ABB RAPID module: Module1.mod

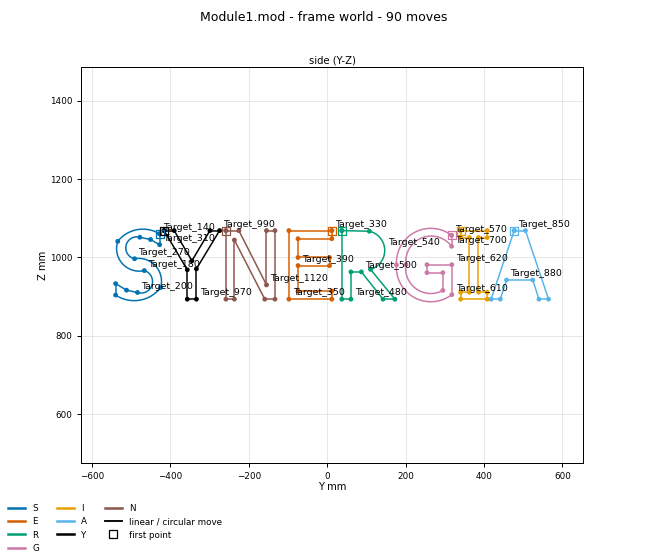
[picture p0: tool path of Module1.mod in frame world, 90 of 90 moves have a stored position in this frame; points joined in program order, loops and branches not executed]
MODULE Module1
	CONST robtarget Target_140:=[[750,-427.603905619,1060.300093764],[0,0,0.978993144,-0.20389317],[0,0,0,0],[9E9,9E9,9E9,9E9,9E9,9E9]];
	CONST robtarget Target_150:=[[750,-479.650096867,1071.645312565],[0,0,0.978993144,-0.20389317],[0,0,0,0],[9E9,9E9,9E9,9E9,9E9,9E9]];
	CONST robtarget Target_160:=[[750,-534.355323771,1041.137310133],[0,0,0.978993144,-0.20389317],[0,0,0,0],[9E9,9E9,9E9,9E9,9E9,9E9]];
	CONST robtarget Target_170:=[[750,-527.158200594,989.9597372],[0,0,0.978993144,-0.20389317],[0,0,0,0],[9E9,9E9,9E9,9E9,9E9,9E9]];
	CONST robtarget Target_180:=[[750,-466.603095246,966.560223424],[0,0,0.978993144,-0.20389317],[0,0,0,0],[9E9,9E9,9E9,9E9,9E9,9E9]];
	CONST robtarget Target_190:=[[750,-447.511219233,927.862391171],[0,0,0.978993144,-0.20389317],[0,0,0,0],[9E9,9E9,9E9,9E9,9E9,9E9]];
	CONST robtarget Target_200:=[[750,-484.046369152,910.543205595],[0,0,0.978993144,-0.20389317],[0,0,0,0],[9E9,9E9,9E9,9E9,9E9,9E9]];
	CONST robtarget Target_210:=[[750,-512.054878066,916.499445466],[0,0,0.978993144,-0.20389317],[0,0,0,0],[9E9,9E9,9E9,9E9,9E9,9E9]];
	CONST robtarget Target_220:=[[750,-539.77975651,933.233643197],[0,0,0.978993144,-0.20389317],[0,0,0,0],[9E9,9E9,9E9,9E9,9E9,9E9]];
	CONST robtarget Target_230:=[[750,-539.77975651,904.019704785],[0,0,0.978993144,-0.20389317],[0,0,0,0],[9E9,9E9,9E9,9E9,9E9,9E9]];
	CONST robtarget Target_240:=[[750,-482.344586332,890.405442224],[0,0,0.978993144,-0.20389317],[0,0,0,0],[9E9,9E9,9E9,9E9,9E9,9E9]];
	CONST robtarget Target_250:=[[750,-424.980323771,923.164761511],[0,0,0.978993144,-0.20389317],[0,0,0,0],[9E9,9E9,9E9,9E9,9E9,9E9]];
	CONST robtarget Target_260:=[[750,-439.941831064,980.617658594],[0,0,0.978993144,-0.20389317],[0,0,0,0],[9E9,9E9,9E9,9E9,9E9,9E9]];
	CONST robtarget Target_270:=[[750,-491.420761372,996.76686848],[0,0,0.978993144,-0.20389317],[0,0,0,0],[9E9,9E9,9E9,9E9,9E9,9E9]];
	CONST robtarget Target_280:=[[750,-511.753520692,1035.145616454],[0,0,0.978993144,-0.20389317],[0,0,0,0],[9E9,9E9,9E9,9E9,9E9,9E9]];
	CONST robtarget Target_290:=[[750,-478.090129282,1051.507549193],[0,0,0.978993144,-0.20389317],[0,0,0,0],[9E9,9E9,9E9,9E9,9E9,9E9]];
	CONST robtarget Target_300:=[[750,-450.719788925,1045.834939793],[0,0,0.978993144,-0.20389317],[0,0,0,0],[9E9,9E9,9E9,9E9,9E9,9E9]];
	CONST robtarget Target_310:=[[750,-427.603905619,1032.504307702],[0,0,0.978993144,-0.20389317],[0,0,0,0],[9E9,9E9,9E9,9E9,9E9,9E9]];
	CONST robtarget Target_320:=[[750,-427.603905619,1060.300093764],[0,0,0.978993144,-0.20389317],[0,0,0,0],[9E9,9E9,9E9,9E9,9E9,9E9]];
	CONST robtarget Target_330:=[[750,11.739692436,1068.525377394],[0,0,0.982498266,0.18627173],[0,-1,0,0],[9E9,9E9,9E9,9E9,9E9,9E9]];
	CONST robtarget Target_340:=[[750,-97.74166899,1068.525377394],[0,0,0.982498266,0.18627173],[-1,-2,0,1],[9E9,9E9,9E9,9E9,9E9,9E9]];
	CONST robtarget Target_350:=[[750,-97.74166899,893.525377394],[0,0,0.982498266,0.18627173],[-1,1,1,0],[9E9,9E9,9E9,9E9,9E9,9E9]];
	CONST robtarget Target_360:=[[750,11.739692436,893.525377394],[0,0,0.982498266,0.18627173],[0,-2,1,0],[9E9,9E9,9E9,9E9,9E9,9E9]];
	CONST robtarget Target_370:=[[750,11.739692436,914.230401706],[0,0,0.982498266,0.18627173],[0,-2,1,0],[9E9,9E9,9E9,9E9,9E9,9E9]];
	CONST robtarget Target_380:=[[750,-74.483970449,914.230401706],[0,0,0.982498266,0.18627173],[-1,1,1,0],[9E9,9E9,9E9,9E9,9E9,9E9]];
	CONST robtarget Target_390:=[[750,-74.483970449,979.181779339],[0,0,0.982498266,0.18627173],[-1,1,1,0],[9E9,9E9,9E9,9E9,9E9,9E9]];
	CONST robtarget Target_400:=[[750,5.925267801,979.181779339],[0,0,0.982498266,0.18627173],[0,-2,1,0],[9E9,9E9,9E9,9E9,9E9,9E9]];
	CONST robtarget Target_410:=[[750,5.925267801,999.88680365],[0,0,0.982498266,0.18627173],[0,-2,1,0],[9E9,9E9,9E9,9E9,9E9,9E9]];
	CONST robtarget Target_420:=[[750,-74.483970449,999.88680365],[0,0,0.982498266,0.18627173],[-1,1,2,0],[9E9,9E9,9E9,9E9,9E9,9E9]];
	CONST robtarget Target_430:=[[750,-74.483970449,1047.820353083],[0,0,0.982498266,0.18627173],[-1,1,-2,0],[9E9,9E9,9E9,9E9,9E9,9E9]];
	CONST robtarget Target_440:=[[750,11.739692436,1047.820353083],[0,0,0.982498266,0.18627173],[0,0,-2,1],[9E9,9E9,9E9,9E9,9E9,9E9]];
	CONST robtarget Target_450:=[[750,11.739692436,1068.525377394],[0,0,0.982498266,0.18627173],[0,1,-2,1],[9E9,9E9,9E9,9E9,9E9,9E9]];
	CONST robtarget Target_460:=[[750,37.266434738,1068.525377394],[0,0,0.978993144,-0.20389317],[0,0,0,0],[9E9,9E9,9E9,9E9,9E9,9E9]];
	CONST robtarget Target_470:=[[750,37.266434738,893.525377394],[0,0,0.978993144,-0.20389317],[0,0,0,0],[9E9,9E9,9E9,9E9,9E9,9E9]];
	CONST robtarget Target_480:=[[750,60.524133279,893.525377394],[0,0,0.978993144,-0.20389317],[0,0,0,0],[9E9,9E9,9E9,9E9,9E9,9E9]];
	CONST robtarget Target_490:=[[750,60.524133279,963.156657783],[0,0,0.978993144,-0.20389317],[0,0,0,0],[9E9,9E9,9E9,9E9,9E9,9E9]];
	CONST robtarget Target_500:=[[750,87.185397461,963.156657783],[0,0,0.978993144,-0.20389317],[0,0,0,0],[9E9,9E9,9E9,9E9,9E9,9E9]];
	CONST robtarget Target_510:=[[750,142.493339114,893.525377394],[0,0,0.978993144,-0.20389317],[0,0,0,0],[9E9,9E9,9E9,9E9,9E9,9E9]];
	CONST robtarget Target_520:=[[750,172.699984171,893.525377394],[0,0,0.978993144,-0.20389317],[0,0,0,0],[9E9,9E9,9E9,9E9,9E9,9E9]];
	CONST robtarget Target_530:=[[750,110.443096002,969.680158594],[0,0,0.978993144,-0.20389317],[0,0,0,0],[9E9,9E9,9E9,9E9,9E9,9E9]];
	CONST robtarget Target_540:=[[750,146.747796164,1021.017273667],[0,0,0.978993144,-0.20389317],[0,0,0,0],[9E9,9E9,9E9,9E9,9E9,9E9]];
	CONST robtarget Target_550:=[[750,107.535883684,1066.894502192],[0,0,0.978993144,-0.20389317],[0,0,0,0],[9E9,9E9,9E9,9E9,9E9,9E9]];
	CONST robtarget Target_560:=[[750,37.266434738,1068.525377394],[0,0,0.978993144,-0.20389317],[0,0,0,0],[9E9,9E9,9E9,9E9,9E9,9E9]];
	CONST robtarget Target_570:=[[750,317.351523879,1056.612897654],[0,0,0.978993144,-0.20389317],[0,0,0,0],[9E9,9E9,9E9,9E9,9E9,9E9]];
	CONST robtarget Target_580:=[[750,225.880697299,1065.405442224],[0,0,0.978993144,-0.20389317],[0,0,0,0],[9E9,9E9,9E9,9E9,9E9,9E9]];
	CONST robtarget Target_590:=[[750,176.670810751,981.167192629],[0,0,0.978993144,-0.20389317],[0,0,0,0],[9E9,9E9,9E9,9E9,9E9,9E9]];
	CONST robtarget Target_600:=[[750,225.951604916,895.794421155],[0,0,0.978993144,-0.20389317],[0,0,0,0],[9E9,9E9,9E9,9E9,9E9,9E9]];
	CONST robtarget Target_610:=[[750,318.060600054,905.154226665],[0,0,0.978993144,-0.20389317],[0,0,0,0],[9E9,9E9,9E9,9E9,9E9,9E9]];
	CONST robtarget Target_620:=[[750,318.060600054,981.592638334],[0,0,0.978993144,-0.20389317],[0,0,0,0],[9E9,9E9,9E9,9E9,9E9,9E9]];
	CONST robtarget Target_630:=[[750,254.52737477,981.592638334],[0,0,0.978993144,-0.20389317],[0,0,0,0],[9E9,9E9,9E9,9E9,9E9,9E9]];
	CONST robtarget Target_640:=[[750,254.52737477,961.171244493],[0,0,0.978993144,-0.20389317],[0,0,0,0],[9E9,9E9,9E9,9E9,9E9,9E9]];
	CONST robtarget Target_650:=[[750,295.086531983,961.171244493],[0,0,0.978993144,-0.20389317],[0,0,0,0],[9E9,9E9,9E9,9E9,9E9,9E9]];
	CONST robtarget Target_660:=[[750,295.086531983,915.932184526],[0,0,0.978993144,-0.20389317],[0,0,0,0],[9E9,9E9,9E9,9E9,9E9,9E9]];
	CONST robtarget Target_670:=[[750,235.098687574,915.010385498],[0,0,0.978993144,-0.20389317],[0,0,0,0],[9E9,9E9,9E9,9E9,9E9,9E9]];
	CONST robtarget Target_680:=[[750,200.921215937,981.876268804],[0,0,0.978993144,-0.20389317],[0,0,0,0],[9E9,9E9,9E9,9E9,9E9,9E9]];
	CONST robtarget Target_690:=[[750,234.531426634,1046.756738821],[0,0,0.978993144,-0.20389317],[0,0,0,0],[9E9,9E9,9E9,9E9,9E9,9E9]];
	CONST robtarget Target_700:=[[750,317.351523879,1028.533481122],[0,0,0.978993144,-0.20389317],[0,0,0,0],[9E9,9E9,9E9,9E9,9E9,9E9]];
	CONST robtarget Target_710:=[[750,317.351523879,1056.612897654],[0,0,0.978993144,-0.20389317],[0,0,0,0],[9E9,9E9,9E9,9E9,9E9,9E9]];
	CONST robtarget Target_720:=[[750,340.467407185,1068.525377394],[0,0,0.978993144,-0.20389317],[0,0,0,0],[9E9,9E9,9E9,9E9,9E9,9E9]];
	CONST robtarget Target_730:=[[750,340.467407185,1050.656657783],[0,0,0.978993144,-0.20389317],[0,0,0,0],[9E9,9E9,9E9,9E9,9E9,9E9]];
	CONST robtarget Target_740:=[[750,362.732399081,1050.656657783],[0,0,0.978993144,-0.20389317],[0,0,0,0],[9E9,9E9,9E9,9E9,9E9,9E9]];
	CONST robtarget Target_750:=[[750,362.732399081,911.394097005],[0,0,0.978993144,-0.20389317],[0,0,0,0],[9E9,9E9,9E9,9E9,9E9,9E9]];
	CONST robtarget Target_760:=[[750,340.467407185,911.394097005],[0,0,0.978993144,-0.20389317],[0,0,0,0],[9E9,9E9,9E9,9E9,9E9,9E9]];
	CONST robtarget Target_770:=[[750,340.467407185,893.525377394],[0,0,0.978993144,-0.20389317],[0,0,0,0],[9E9,9E9,9E9,9E9,9E9,9E9]];
	CONST robtarget Target_780:=[[750,408.255089519,893.525377394],[0,0,0.978993144,-0.20389317],[0,0,0,0],[9E9,9E9,9E9,9E9,9E9,9E9]];
	CONST robtarget Target_790:=[[750,408.255089519,911.394097005],[0,0,0.978993144,-0.20389317],[0,0,0,0],[9E9,9E9,9E9,9E9,9E9,9E9]];
	CONST robtarget Target_800:=[[750,385.990097623,911.394097005],[0,0,0.978993144,-0.20389317],[0,0,0,0],[9E9,9E9,9E9,9E9,9E9,9E9]];
	CONST robtarget Target_810:=[[750,385.990097623,1050.656657783],[0,0,0.978993144,-0.20389317],[0,0,0,0],[9E9,9E9,9E9,9E9,9E9,9E9]];
	CONST robtarget Target_820:=[[750,408.255089519,1050.656657783],[0,0,0.978993144,-0.20389317],[0,0,0,0],[9E9,9E9,9E9,9E9,9E9,9E9]];
	CONST robtarget Target_830:=[[750,408.255089519,1068.525377394],[0,0,0.978993144,-0.20389317],[0,0,0,0],[9E9,9E9,9E9,9E9,9E9,9E9]];
	CONST robtarget Target_840:=[[750,340.467407185,1068.525377394],[0,0,0.978993144,-0.20389317],[0,0,0,0],[9E9,9E9,9E9,9E9,9E9,9E9]];
	CONST robtarget Target_850:=[[750,477.177293733,1068.525377394],[0,0,0.978993144,-0.20389317],[0,0,0,0],[9E9,9E9,9E9,9E9,9E9,9E9]];
	CONST robtarget Target_860:=[[750,418.18215597,893.525377394],[0,0,0.978993144,-0.20389317],[0,0,0,0],[9E9,9E9,9E9,9E9,9E9,9E9]];
	CONST robtarget Target_870:=[[750,441.723484981,893.525377394],[0,0,0.978993144,-0.20389317],[0,0,0,0],[9E9,9E9,9E9,9E9,9E9,9E9]];
	CONST robtarget Target_880:=[[750,457.606791302,942.451633472],[0,0,0.978993144,-0.20389317],[0,0,0,0],[9E9,9E9,9E9,9E9,9E9,9E9]];
	CONST robtarget Target_890:=[[750,524.401766991,942.451633472],[0,0,0.978993144,-0.20389317],[0,0,0,0],[9E9,9E9,9E9,9E9,9E9,9E9]];
	CONST robtarget Target_900:=[[750,540.285073312,893.525377394],[0,0,0.978993144,-0.20389317],[0,0,0,0],[9E9,9E9,9E9,9E9,9E9,9E9]];
	CONST robtarget Target_910:=[[750,564.819108968,893.525377394],[0,0,0.978993144,-0.20389317],[0,0,0,0],[9E9,9E9,9E9,9E9,9E9,9E9]];
	CONST robtarget Target_920:=[[750,505.823971205,1068.525377394],[0,0,0.978993144,-0.20389317],[0,0,0,0],[9E9,9E9,9E9,9E9,9E9,9E9]];
	CONST robtarget Target_930:=[[750,477.177293733,1068.525377394],[0,0,0.978993144,-0.20389317],[0,0,0,0],[9E9,9E9,9E9,9E9,9E9,9E9]];
	CONST robtarget Target_940:=[[750,-416.116871583,1068.525377394],[0,0,0.978993144,-0.20389317],[0,0,0,0],[9E9,9E9,9E9,9E9,9E9,9E9]];
	CONST robtarget Target_950:=[[750,-356.979918585,968.545636714],[0,0,0.978993144,-0.20389317],[0,0,0,0],[9E9,9E9,9E9,9E9,9E9,9E9]];
	CONST robtarget Target_960:=[[750,-356.979918585,893.525377394],[0,0,0.978993144,-0.20389317],[0,0,0,0],[9E9,9E9,9E9,9E9,9E9,9E9]];
	CONST robtarget Target_970:=[[750,-333.722220043,893.525377394],[0,0,0.978993144,-0.20389317],[0,0,0,0],[9E9,9E9,9E9,9E9,9E9,9E9]];
	CONST robtarget Target_980:=[[750,-333.722220043,970.956495709],[0,0,0.978993144,-0.20389317],[0,0,0,0],[9E9,9E9,9E9,9E9,9E9,9E9]];
	CONST robtarget Target_990:=[[750,-274.585267045,1068.525377394],[0,0,0.978993144,-0.20389317],[0,0,0,0],[9E9,9E9,9E9,9E9,9E9,9E9]];
	CONST robtarget Target_1000:=[[750,-299.261117936,1068.525377394],[0,0,0.978993144,-0.20389317],[0,0,0,0],[9E9,9E9,9E9,9E9,9E9,9E9]];
	CONST robtarget Target_1010:=[[750,-345.209254079,991.519704785],[0,0,0.978993144,-0.20389317],[0,0,0,0],[9E9,9E9,9E9,9E9,9E9,9E9]];
	CONST robtarget Target_1020:=[[750,-390.306498812,1068.525377394],[0,0,0.978993144,-0.20389317],[0,0,0,0],[9E9,9E9,9E9,9E9,9E9,9E9]];
	CONST robtarget Target_1030:=[[750,-416.116871583,1068.525377394],[0,0,0.978993144,-0.20389317],[0,0,0,0],[9E9,9E9,9E9,9E9,9E9,9E9]];
	CONST robtarget Target_1040:=[[750,-258.418330254,1068.525377394],[0,0,0.978993144,-0.20389317],[-1,0,-2,0],[9E9,9E9,9E9,9E9,9E9,9E9]];
	CONST robtarget Target_1050:=[[750,-258.418330254,893.525377394],[0,0,0.978993144,-0.20389317],[0,0,0,0],[9E9,9E9,9E9,9E9,9E9,9E9]];
	CONST robtarget Target_1060:=[[750,-236.720599298,893.525377394],[0,0,0.978993144,-0.20389317],[0,0,0,0],[9E9,9E9,9E9,9E9,9E9,9E9]];
	CONST robtarget Target_1070:=[[750,-236.720599298,1044.416787443],[0,0,0.978993144,-0.20389317],[0,0,0,0],[9E9,9E9,9E9,9E9,9E9,9E9]];
	CONST robtarget Target_1080:=[[750,-159.289480983,893.525377394],[0,0,0.978993144,-0.20389317],[0,0,0,0],[9E9,9E9,9E9,9E9,9E9,9E9]];
	CONST robtarget Target_1090:=[[750,-133.195477742,893.525377394],[0,0,0.978993144,-0.20389317],[0,0,0,0],[9E9,9E9,9E9,9E9,9E9,9E9]];
	CONST robtarget Target_1100:=[[750,-133.195477742,1068.525377394],[0,0,0.978993144,-0.20389317],[0,0,0,0],[9E9,9E9,9E9,9E9,9E9,9E9]];
	CONST robtarget Target_1110:=[[750,-154.893208698,1068.525377394],[0,0,0.978993144,-0.20389317],[0,0,0,0],[9E9,9E9,9E9,9E9,9E9,9E9]];
	CONST robtarget Target_1120:=[[750,-154.893208698,929.971892791],[0,0,0.978993144,-0.20389317],[0,0,0,0],[9E9,9E9,9E9,9E9,9E9,9E9]];
	CONST robtarget Target_1130:=[[750,-225.375380497,1068.525377394],[0,0,0.978993144,-0.20389317],[0,0,0,0],[9E9,9E9,9E9,9E9,9E9,9E9]];
	CONST robtarget Target_1140:=[[750,-258.418330254,1068.525377394],[0,0,0.978993144,-0.20389317],[0,0,0,0],[9E9,9E9,9E9,9E9,9E9,9E9]];
	PROC S()
        ConfL \Off;
	    MoveJ Target_140,v1000,fine,Pen_TCP\WObj:=WS;
        StopMove;
        WaitTime 1;
        StartMove;
	    MoveC Target_150,Target_160,v1000,z100,Pen_TCP\WObj:=WS;
	    MoveC Target_170,Target_180,v1000,z100,Pen_TCP\WObj:=WS;
	    MoveC Target_190,Target_200,v1000,z100,Pen_TCP\WObj:=WS;
	    MoveL Target_210,v1000,z100,Pen_TCP\WObj:=WS;
	    MoveL Target_220,v1000,z100,Pen_TCP\WObj:=WS;
	    MoveL Target_230,v1000,z100,Pen_TCP\WObj:=WS;
	    MoveC Target_240,Target_250,v1000,z100,Pen_TCP\WObj:=WS;
	    MoveC Target_260,Target_270,v1000,z100,Pen_TCP\WObj:=WS;
	    MoveC Target_280,Target_290,v1000,z100,Pen_TCP\WObj:=WS;
	    MoveL Target_300,v1000,z100,Pen_TCP\WObj:=WS;
	    MoveL Target_310,v1000,z100,Pen_TCP\WObj:=WS;
	    MoveL Target_320,v1000,z100,Pen_TCP\WObj:=WS;
	ENDPROC
	PROC E()
	    MoveL Target_330,v1000,z100,Pen_TCP\WObj:=WE;
	    MoveL Target_340,v1000,z100,Pen_TCP\WObj:=WE;
	    MoveL Target_350,v1000,z100,Pen_TCP\WObj:=WE;
	    MoveL Target_360,v1000,z100,Pen_TCP\WObj:=WE;
	    MoveL Target_370,v1000,z100,Pen_TCP\WObj:=WE;
	    MoveL Target_380,v1000,z100,Pen_TCP\WObj:=WE;
	    MoveL Target_390,v1000,z100,Pen_TCP\WObj:=WE;
	    MoveL Target_400,v1000,z100,Pen_TCP\WObj:=WE;
	    MoveL Target_410,v1000,z100,Pen_TCP\WObj:=WE;
	    MoveL Target_420,v1000,z100,Pen_TCP\WObj:=WE;
	    MoveL Target_430,v1000,z100,Pen_TCP\WObj:=WE;
	    MoveL Target_440,v1000,z100,Pen_TCP\WObj:=WE;
	    MoveL Target_450,v1000,z100,Pen_TCP\WObj:=WE;
	ENDPROC
	PROC R()
	    MoveL Target_460,v1000,z100,Pen_TCP\WObj:=WR;
	    MoveL Target_470,v1000,z100,Pen_TCP\WObj:=WR;
	    MoveL Target_480,v1000,z100,Pen_TCP\WObj:=WR;
	    MoveL Target_490,v1000,z100,Pen_TCP\WObj:=WR;
	    MoveL Target_500,v1000,z100,Pen_TCP\WObj:=WR;
	    MoveL Target_510,v1000,z100,Pen_TCP\WObj:=WR;
	    MoveL Target_520,v1000,z100,Pen_TCP\WObj:=WR;
	    MoveL Target_530,v1000,z100,Pen_TCP\WObj:=WR;
	    MoveC Target_540,Target_550,v1000,z100,Pen_TCP\WObj:=WR;
	    MoveL Target_560,v1000,z100,Pen_TCP\WObj:=WR;
	ENDPROC
	PROC G()
	    MoveL Target_570,v1000,z100,Pen_TCP\WObj:=WG;
	    MoveC Target_580,Target_590,v1000,z100,Pen_TCP\WObj:=WG;
	    MoveC Target_600,Target_610,v1000,z100,Pen_TCP\WObj:=WG;
	    MoveL Target_620,v1000,z100,Pen_TCP\WObj:=WG;
	    MoveL Target_630,v1000,z100,Pen_TCP\WObj:=WG;
	    MoveL Target_640,v1000,z100,Pen_TCP\WObj:=WG;
	    MoveL Target_650,v1000,z100,Pen_TCP\WObj:=WG;
	    MoveL Target_660,v1000,z100,Pen_TCP\WObj:=WG;
	    MoveC Target_670,Target_680,v1000,z100,Pen_TCP\WObj:=WG;
	    MoveC Target_690,Target_700,v1000,z100,Pen_TCP\WObj:=WG;
	    MoveL Target_710,v1000,z100,Pen_TCP\WObj:=WG;
	ENDPROC
	PROC I()
	    MoveL Target_720,v1000,z100,Pen_TCP\WObj:=WI;
	    MoveL Target_730,v1000,z100,Pen_TCP\WObj:=WI;
	    MoveL Target_740,v1000,z100,Pen_TCP\WObj:=WI;
	    MoveL Target_750,v1000,z100,Pen_TCP\WObj:=WI;
	    MoveL Target_760,v1000,z100,Pen_TCP\WObj:=WI;
	    MoveL Target_770,v1000,z100,Pen_TCP\WObj:=WI;
	    MoveL Target_780,v1000,z100,Pen_TCP\WObj:=WI;
	    MoveL Target_790,v1000,z100,Pen_TCP\WObj:=WI;
	    MoveL Target_800,v1000,z100,Pen_TCP\WObj:=WI;
	    MoveL Target_810,v1000,z100,Pen_TCP\WObj:=WI;
	    MoveL Target_820,v1000,z100,Pen_TCP\WObj:=WI;
	    MoveL Target_830,v1000,z100,Pen_TCP\WObj:=WI;
	    MoveL Target_840,v1000,z100,Pen_TCP\WObj:=WI;
	ENDPROC
	PROC A()
	    MoveL Target_850,v1000,z100,Pen_TCP\WObj:=WA;
	    MoveL Target_860,v1000,z100,Pen_TCP\WObj:=WA;
	    MoveL Target_870,v1000,z100,Pen_TCP\WObj:=WA;
	    MoveL Target_880,v1000,z100,Pen_TCP\WObj:=WA;
	    MoveL Target_890,v1000,z100,Pen_TCP\WObj:=WA;
	    MoveL Target_900,v1000,z100,Pen_TCP\WObj:=WA;
	    MoveL Target_910,v1000,z100,Pen_TCP\WObj:=WA;
	    MoveL Target_920,v1000,z100,Pen_TCP\WObj:=WA;
	    MoveL Target_930,v1000,z100,Pen_TCP\WObj:=WA;
	ENDPROC
	PROC Y()
	    MoveL Target_940,v1000,z100,Pen_TCP\WObj:=WY;
	    MoveL Target_950,v1000,z100,Pen_TCP\WObj:=WY;
	    MoveL Target_960,v1000,z100,Pen_TCP\WObj:=WY;
	    MoveL Target_970,v1000,z100,Pen_TCP\WObj:=WY;
	    MoveL Target_980,v1000,z100,Pen_TCP\WObj:=WY;
	    MoveL Target_990,v1000,z100,Pen_TCP\WObj:=WY;
	    MoveL Target_1000,v1000,z100,Pen_TCP\WObj:=WY;
	    MoveL Target_1010,v1000,z100,Pen_TCP\WObj:=WY;
	    MoveL Target_1020,v1000,z100,Pen_TCP\WObj:=WY;
	    MoveL Target_1030,v1000,z100,Pen_TCP\WObj:=WY;
	ENDPROC
	PROC N()
	    MoveL Target_1040,v1000,z100,Pen_TCP\WObj:=WN;
	    MoveL Target_1050,v1000,z100,Pen_TCP\WObj:=WN;
	    MoveL Target_1060,v1000,z100,Pen_TCP\WObj:=WN;
	    MoveL Target_1070,v1000,z100,Pen_TCP\WObj:=WN;
	    MoveL Target_1080,v1000,z100,Pen_TCP\WObj:=WN;
	    MoveL Target_1090,v1000,z100,Pen_TCP\WObj:=WN;
	    MoveL Target_1100,v1000,z100,Pen_TCP\WObj:=WN;
	    MoveL Target_1110,v1000,z100,Pen_TCP\WObj:=WN;
	    MoveL Target_1120,v1000,z100,Pen_TCP\WObj:=WN;
	    MoveL Target_1130,v1000,z100,Pen_TCP\WObj:=WN;
	    MoveL Target_1140,v1000,z100,Pen_TCP\WObj:=WN;

    PROC rDoExit()
        STOP;
    ENDPROC

ENDMODULE
